(*********************************** G.D S.p.A. - Technical Department ***********************************
============= PROGRAM INFO ============
FOLDER:             TBD
MACHINES INVOLVED:  TBD 

============= DESCRIPTION =============
csp machine declaration

============= REVISIONS ===============
Date		Version	 	Author      	Description             
----------	-------		------------  	--------------------------------------------
2019/04/05 	0000.00	 	M.Grasso		Creation of the PRG

**********************************************************************************************************)
(*$R process_ref := prc; $*)
PROGRAM csp_case_closing_ls_lower
VAR
	
	prc:												process;
	prc_path:											STRING;
	
	fsm_enable_condition:								BOOL := FALSE;
	fsm_next_status:									csp_case_closing_status_enum;
	fsm_status:											csp_case_closing_status_enum;
	
	axis:												axis;
	phase_velocity_degps:								LREAL := 20.0;
	phase_done:											BOOL;
	axis_calculate_cam_slave_master_position_deg:		LREAL := 0.0;
	axis_calculated_cam_slave_position_deg:				LREAL := 0.0;
	slave_position_has_been_calculated:					BOOL  := FALSE;
	phase_enable:										BOOL:=TRUE;
	engage_enable:										BOOL:=TRUE;
	disable_req:										BOOL:=FALSE;
	debug_state_machine:								BOOL:=FALSE;
	debug_state_machine_one_step:						BOOL:=FALSE;
	cam_id:												INT := CASE_CLOSING_LOWER_RUN_CAM;
	slave_scaling:										LREAL := 1; (*$P $*)
	master_scaling:										LREAL := 1;
	master_offset:										LREAL := 315; (*$P $*)
	slave_offset:										LREAL := -25;  (*$P $*)
	
	in_accu_safe_pos:                                   BOOL := FALSE;
    accu_safe_pos:                                      LREAL := 267;
	accu_tolerance: 									LREAL := 5;
	
	torque_limit:										INT := 2000;    (*$P $*)
	torque_limit_old:									INT;

	Closing_Lower_RFID_Check_Done: 						BOOL := FALSE;
	RFID_check_pos: 									LREAL := 344;
	rfid_fake: 											BOOL := false;

	servo_on_condition: 								BOOL;
	enable_delay: 										TON;
	Torque_force_constant: 								LREAL := 0.47;
END_VAR

VAR CONSTANT
	(*Just in case you prefer having constants instead of numbers*)
	MOTOR_MAX_VELOCITY_DEGPS:							LREAL := 9600;
	MOTOR_MAX_ACCELLERATION_DEGPS2:						LREAL := 4800;
	MOTOR_MAX_DECELLERATION_DEGPS2:						LREAL := 4800;
	MOTOR_MAX_JERK_DEGPS3:								LREAL := 100000000; 
	MOTOR_MAX_FOLLOWING_ERROR_DEG:						LREAL := 5;
END_VAR

_read_var_input();

_object_manager();

IF NOT objects_running()
THEN
	RETURN;	
END_IF

_read_process_image();

_mode_manager();

CASE process_get_mode(prc) OF
	MODE_ABSENT:
		IF axis_get_mode(axis) = MODE_TEST
		THEN
			safety_integrated_series_close(csp_case_main_safety_drives_SD2500.chA_smes_sis);
		END_IF
		RETURN;
	MODE_INACTIVE:
		RETURN;
	MODE_TEST:
		_handle_process_test();
END_CASE

_set_runtime_properties();

(********************************* BODY *********************************)
axis.actual_torque := (axis.actual_current * Torque_force_constant)/1000;

//Checks if axis position is within the acc-u-change safe position
IF 	ABS(axis.actual_position - accu_safe_pos)  < accu_tolerance
	OR (360 - axis.actual_position) < accu_tolerance
THEN
	in_accu_safe_pos := TRUE;
ELSE
	in_accu_safe_pos := FALSE;   
END_IF

// Sets the torque limit
IF torque_limit <> Torque_limit_old
	THEN
	 IF soe_drive_channel_write_parameter(
			channel:=csp_case_closing_ls_lower.axis.soe_drive_channel, 
			idn:= S_0_IDN + 92, 
			data_element:=soe_drive_element_value , 
			data_source:= ADR(torque_limit), 
			data_lenght:= SIZEOF(torque_limit), 
			CONVERSION_this:= csp_case_closing_ls_lower.axis.soe_drive^) = SOE_DRIVE_RETURN_VALUE_DONE
	THEN		
		torque_limit_old := Torque_limit;
	END_IF	
END_IF

(* MACHINE COMMANDS *)
fsm_enable_condition := axis_is_ok(FALSE, axis)
						AND
						process_is_ready(prc)
						AND
						process_subtree_is_ready(prc)
						AND						
						(csp_main_motorization.motorization_axis_redefined_at_powerup OR csp_main_accuchange.Brand_Change_Occurred)
						AND
						servo_on_condition
						AND
						NOT jog_manager_is_jog_axis_active(SMTR2503_CASE_CLOSING_LS_LOWER, csp_main_jogManager.jog_manager_real)						
						AND
						NOT disable_req;

IF	(NOT fsm_enable_condition
	OR
	disable_req)
	AND
	fsm_status <> CSP_CASE_CLOSING_STATUS_DISABLED
	AND
	fsm_status < CSP_CASE_CLOSING_STATUS_STOP_REQUEST
THEN
	fsm_status	:=	CSP_CASE_CLOSING_STATUS_DISABLE_REQUEST;
END_IF


CASE fsm_status OF
	
	CSP_CASE_CLOSING_STATUS_NOT_INITIALIZED:
       
		IF	axis_is_ok(return_when_absent := TRUE, CONVERSION_this := axis)
        THEN
            fsm_next_status := CSP_CASE_CLOSING_STATUS_DISABLED;
        END_IF

		
	CSP_CASE_CLOSING_STATUS_DISABLED:

		phase_done := FALSE;
	
		IF	fsm_enable_condition
			AND
			(
			(motorization_manager_is_starting(csp_main_motorization_manager.motm))
			OR
			jog_manager_is_jog_axis_active(JOG_LIST_CSP_CASE_TRANSPORT_VIRTUAL, csp_main_jogManager.jog_manager_virtual)
			OR
			jog_manager_is_jog_axis_active(JOG_LIST_CSP_CASE_VIRTUAL, csp_main_jogManager.jog_manager_virtual)	
			)
		THEN
			debug_state_machine :=FALSE;
			fsm_next_status := CSP_CASE_CLOSING_STATUS_ENABLE_REQUEST;
		END_IF;

		
	CSP_CASE_CLOSING_STATUS_ENABLE_REQUEST:
		
		axis_enable(axis);
		IF axis_is_standstill(axis)
		THEN
			fsm_next_status	:=	CSP_CASE_CLOSING_STATUS_ENABLED;
		END_IF;		

		
	CSP_CASE_CLOSING_STATUS_ENABLED:
		
		IF NOT csp_main_accuChange.machine_size_complete
		THEN
			fsm_next_status    := CSP_CASE_CLOSING_STATUS_CHANGE_OVER_MODE;
		ELSE   
			fsm_next_status    := CSP_CASE_CLOSING_STATUS_HOME_REQUEST;
		END_IF
   
		
	CSP_CASE_CLOSING_STATUS_CHANGE_OVER_MODE:
			
		//During size change the paddles move down to the the safe position
		IF axis_move_absolute(
            position         := accu_safe_pos, 
            velocity         := phase_velocity_degps,
            direction        := AXIS_SHORTEST_WAY,
            acceleration     := MOTOR_MAX_ACCELLERATION_DEGPS2,
            deceleration     := MOTOR_MAX_DECELLERATION_DEGPS2,
            jerk             := MOTOR_MAX_JERK_DEGPS3,
            buffer_mode     := AXIS_BUFFER_MODE_BUFFERED,
            CONVERSION_this := axis)  
  		THEN
			IF axis_is_absolute_moving(axis)
			THEN
				fsm_next_status := CSP_CASE_CLOSING_STATUS_CHANGE_OVER_MODE_MOVE_DONE;
			END_IF
		END_IF
		
		
	CSP_CASE_CLOSING_STATUS_CHANGE_OVER_MODE_MOVE_DONE:
	
		IF 	csp_main_accuChange.Motion_Motors_New_Size_Req
			AND axis_is_standstill(axis)
		THEN
			fsm_next_status	:=	CSP_CASE_CLOSING_STATUS_HOME_REQUEST;
		END_IF;
	
		
	CSP_CASE_CLOSING_STATUS_HOME_REQUEST: 
	
		Closing_Lower_RFID_Check_Done := FALSE;
		fsm_next_status	:=	CSP_CASE_CLOSING_STATUS_HOME_DONE;

		
	CSP_CASE_CLOSING_STATUS_HOMING:

		axis.home.done := TRUE;
		IF axis_home_done(axis)
		THEN
			fsm_next_status	:=	CSP_CASE_CLOSING_STATUS_HOME_DONE;
		END_IF

		
	CSP_CASE_CLOSING_STATUS_HOME_DONE:
	
		IF phase_enable
		THEN
			fsm_next_status	:= CSP_CASE_CLOSING_STATUS_CALCULATE_SLAVE_POSITION_REQUEST;
		END_IF
		
	
	CSP_CASE_CLOSING_STATUS_CALCULATE_SLAVE_POSITION_REQUEST:

		axis_calculate_cam_slave_master_position_deg := 
		LMOD	(axis_get_actual_modulo_position(csp_case_transport_virtualMaster.axis) (*master axis*)
	             	+
		(master_offset ), (*initialized at 0° position*)
			G_MODULO_360_DEG);	(*master_scaling and slave_scaling initialized at 360° since the cams are normed in a range equal to 0-1.*)
		IF axis_calculate_cam_slave_dynamics_data(
				cam_id := cam_id,
				master_scaling := master_scaling,
				master_position := axis_calculate_cam_slave_master_position_deg,
				slave_scaling := slave_scaling,
				CONVERSION_this := axis)
		THEN
			fsm_next_status := CSP_CASE_CLOSING_STATUS_CALCULATING_SLAVE_POSITION;
		END_IF


	CSP_CASE_CLOSING_STATUS_CALCULATING_SLAVE_POSITION:
		
		IF	axis_cam_slave_dynamics_data_calculated(axis)
		THEN
			(*The “axis_get_cam_slave_dynamics_position” method returns the position of the slave within the cam plate table at the master position calculated for the instance specified: *)
			axis_calculated_cam_slave_position_deg :=(axis_get_cam_slave_dynamics_position(axis) + slave_offset);
			slave_position_has_been_calculated := TRUE;
			fsm_next_status := CSP_CASE_CLOSING_STATUS_PHASE_REQUEST;
		END_IF


	CSP_CASE_CLOSING_STATUS_PHASE_REQUEST:

		IF	axis_is_standstill(axis)
			AND csp_case_closing_ls.phase_lower
		THEN
			axis_move_absolute(
				position 		:= axis_calculated_cam_slave_position_deg,(*calculated above, the slave is moved*)
				velocity 		:= phase_velocity_degps,
				direction		:= AXIS_SHORTEST_WAY,
				acceleration 	:= MOTOR_MAX_ACCELLERATION_DEGPS2,
				deceleration 	:= MOTOR_MAX_DECELLERATION_DEGPS2,
				jerk 			:= MOTOR_MAX_JERK_DEGPS3, 
				buffer_mode 	:= AXIS_BUFFER_MODE_BUFFERED,
				CONVERSION_this 			:= axis
				); 
		END_IF

		IF axis_is_absolute_moving(axis)
		THEN
			fsm_next_status	:=	CSP_CASE_CLOSING_STATUS_PHASING;
		END_IF

		
	CSP_CASE_CLOSING_STATUS_PHASING:

		IF axis_is_standstill(axis)
		THEN
			phase_done := TRUE;
			fsm_next_status	:=	CSP_CASE_CLOSING_STATUS_PHASED;
		END_IF

		
	CSP_CASE_CLOSING_STATUS_PHASED:

		IF engage_enable
		THEN
			fsm_next_status := CSP_CASE_CLOSING_STATUS_CAM_ENGAGED_REQ;
		END_IF


	CSP_CASE_CLOSING_STATUS_CAM_ENGAGED_REQ:
		
		(* WAITS FOR MOVE REQUEST FOR CROSSPUSHER AND CAMS TO CROSSPUSHER VIRTUAL MASTER *)
		axis_engage_cam(
			cam_id 			:= cam_id,
			master_engage_mode 	:= AXIS_CAM_ENGAGE_ABSOLUTE,
			slave_engage_mode 	:= AXIS_CAM_ENGAGE_ABSOLUTE, 
			activation_mode 	:= AXIS_CAM_ACTIVATION_IMMEDIATELY, 
			activation_position	:= 0,
			master_scaling_mode	:= AXIS_CAM_SCALING_MODE_USER_DEFINED,
			slave_scaling_mode	:= AXIS_CAM_SCALING_MODE_USER_DEFINED,
			master_offset 		:= master_offset,	//moved right  respect to the original Y axis of the cam profile
			slave_offset 		:= slave_offset,	
			master_scaling 		:= master_scaling,
			slave_scaling 		:= slave_scaling,
			interpolation_type 		:= AXIS_CAM_INTERPOLATION_SYSTEM_DEFAULT,
			master 			:= csp_case_transport_virtualMaster.axis,
			CONVERSION_this 	:= axis);	
			
		IF	axis_is_cam_engaged(axis)
		THEN
			fsm_next_status := CSP_CASE_CLOSING_STATUS_CAM_ENGAGED;
		END_IF

	
	CSP_CASE_CLOSING_STATUS_AXIS_ENGAGE_VERIFY :
		
		;
		
		
	CSP_CASE_CLOSING_STATUS_CAM_ENGAGED:
	
		IF 	machine_is_stop_emergency_active(csp.mch)
			AND motorization_manager_is_stopped(csp_main_motorization_manager.motm)	
		THEN
			fsm_next_status := CSP_CASE_CLOSING_STATUS_DISENGAGE_REQUEST;
		END_IF
		
		
	CSP_CASE_CLOSING_STATUS_RUNNING:
	
		;
		
		
	CSP_CASE_CLOSING_STATUS_DISENGAGE_REQUEST:

		fsm_next_status := CSP_CASE_CLOSING_STATUS_DISENGAGING;
		
		
	CSP_CASE_CLOSING_STATUS_DISENGAGING:
	
		IF axis_disengage(
			mode:= AXIS_DISENGAGE_AND_ON_PHASE_STOP, 
			position:= 0, 
			velocity:= 100, 
			acceleration:= MOTOR_MAX_ACCELLERATION_DEGPS2, 
			deceleration:= MOTOR_MAX_DECELLERATION_DEGPS2, 
			jerk:= MOTOR_MAX_JERK_DEGPS3, 
			CONVERSION_this:= axis)
		THEN
			fsm_next_status := CSP_CASE_CLOSING_STATUS_CAM_ENGAGED_REQ;
		END_IF
	
		
	CSP_CASE_CLOSING_STATUS_STOP_REQUEST:

		axis_stop(
		    deceleration 	:= MOTOR_MAX_DECELLERATION_DEGPS2,
		    jerk 			:= MOTOR_MAX_JERK_DEGPS3,
		    CONVERSION_this 			:= axis);

		IF 	axis_is_standstill(axis)
			OR
			NOT axis_is_ok(FALSE, axis)
			OR
			axis_is_disabled(axis)
		THEN
			fsm_next_status := CSP_CASE_CLOSING_STATUS_DISABLE_REQUEST;
		END_IF

		
	CSP_CASE_CLOSING_STATUS_DISABLE_REQUEST:
   		
		axis_disable(axis);
   		fsm_next_status := CSP_CASE_CLOSING_STATUS_DISABLING;

	CSP_CASE_CLOSING_STATUS_DISABLING:
        
		IF	axis_is_disabled(axis)
        THEN
            fsm_next_status := CSP_CASE_CLOSING_STATUS_DISABLED;
        END_IF

END_CASE;

IF 	NOT debug_state_machine
	OR
	debug_state_machine_one_step
THEN
	fsm_status := fsm_next_status;
	debug_state_machine_one_step := FALSE;
END_IF
(************************************************************************)

_handle_messages();

_write_output();

ACTION _handle_messages:
;
END_ACTION

ACTION _handle_process_test:
;
END_ACTION

ACTION _mode_manager:
IF process_mode_req_is_pending(prc)
THEN
    process_apply_mode_req_first_step(prc);
    CASE process_get_mode(prc) OF
        MODE_TO_ABSENT:
			;
        MODE_TO_INACTIVE:
			;
        MODE_TO_TEST:
			;
        MODE_TO_OPERATIONAL:
			;
    END_CASE
    process_apply_mode_req_second_step(prc);
END_IF
END_ACTION

ACTION _object_manager:
IF objects_initialization()
THEN
	sub_process_init(
		object_name									:= 'csp_case_closing_ls_lower.prc', 
		process										:= csp_case_closing_ls.prc, 
		CONVERSION_this								:= prc);
		
	prc_path 										:= process_get_path(prc);
	
		(* axis smes *)
	IF csp_main_configurator.Physical_hw
	THEN	
		axis_init(
			object_name								:= CONCAT(prc_path, '_axis'), 
			axis_type								:= AXIS_TYPE_SERVO, 
			encoder_scaling_factor					:= G_SERVO_ENCODER_SCALING_FACTOR_DEGPINC,
			modulo									:= G_MODULO_360_DEG, 
			process									:= prc, 
			CONVERSION_this							:= axis);

		axis_add_safety_integrated_series(
			safety_integrated_series 				:= csp_case_main_safety_drives_SD2500.chA_smes_sis,
			CONVERSION_this							:= axis);
			
		axis_init_absolute_encoder_preset(
			position                                := 0.0,
			CONVERSION_this                         := axis);
	ELSE
		axis_init(
			object_name								:= CONCAT(prc_path, '_axis'), 
			axis_type								:= AXIS_TYPE_VIRTUAL, 
			encoder_scaling_factor					:= G_VIRTUAL_ENCODER_SCALING_FACTOR_DEGPINC,
			modulo									:= G_MODULO_360_DEG, 
			process									:= prc, 
			CONVERSION_this							:= axis);
	END_IF 
		
	axis_set_max_dynamic(
		reference_velocity							:=	MOTOR_MAX_VELOCITY_DEGPS,
		velocity									:=	MOTOR_MAX_VELOCITY_DEGPS,
		acceleration								:=	MOTOR_MAX_ACCELLERATION_DEGPS2,
		deceleration								:=	MOTOR_MAX_DECELLERATION_DEGPS2,
		jerk										:=	MOTOR_MAX_JERK_DEGPS3,
		following_error								:=	MOTOR_MAX_FOLLOWING_ERROR_DEG,
		CONVERSION_this								:=	axis);
	
		
	jog_manager_add_axis(
		list_index									:= SMTR2503_CASE_CLOSING_LS_LOWER,
		axis										:= axis,
		master_axis									:= FALSE,
		jog_type									:= JOG_TYPE_LINEAR,
		sw_limit_positive							:= 800,
		sw_limit_negative							:= 0,
		CONVERSION_this								:= csp_main_jogManager.jog_manager_real);
	
	axis_add_soe_drive(
		channel										:=	SOE_DRIVE_CHANNEL_A,
		soe_drive									:=	csp_case_main_drives.SD2500_drv,
		CONVERSION_this								:=	axis);
		
END_IF
IF objects_running()
THEN
	process_cycle(prc);
	axis_cycle(axis);
END_IF
END_ACTION

ACTION _read_process_image:
;
END_ACTION

ACTION _read_var_input:
disable_req := csp_case.disable_req;
END_ACTION

ACTION _set_runtime_properties:
enable_delay(IN:=axis_is_ready_to_enable(axis) , PT:=T#2S , Q=> servo_on_condition , ET=> );
END_ACTION

ACTION _write_output:
;
END_ACTION

END_PROGRAM

(* stored: Version 1.1.0.1, ProductVersion 3.1.4024.3
   POU csp_case_closing_ls_lower: Id {39069e50-2836-45ac-9fd5-5a5b1ee83f2b}, SpecialFunc None
   Action _handle_messages: Id {b5023d2b-f117-4385-b0e5-ff076e536380}
   Action _handle_process_test: Id {68ff7fa1-8b0c-4f42-ab86-e9d8c394b57e}
   Action _mode_manager: Id {f8bee80f-e8dc-4208-a29e-10b33de0f556}
   Action _object_manager: Id {3c7b6f0c-0690-4542-919d-f467101045c7}
   Action _read_process_image: Id {f6348841-eb7e-4a61-b689-fc29d2a7a0ad}
   Action _read_var_input: Id {98f1bac2-cd29-4776-99dc-149b601e1f0b}
   Action _set_runtime_properties: Id {55fd18d8-7224-4365-b760-e80d08d78b9f}
   Action _write_output: Id {61d22664-5a6e-4818-b315-c9b88a81f38b} *)
